// TIA Portal V19 export
DATA_BLOCK "GBL_TandD_DB"   // DB104
// stored: InstanceOfName GBL_TandD, InstanceOfType FB
"GBL_TandD"
   // VAR
   //    "write time" { ExternalAccessible := 'False'; ExternalVisible := 'False'; ExternalWritable := 'False'} : DTL;
   //    "System Time" { ExternalAccessible := 'False'; ExternalVisible := 'False'; ExternalWritable := 'False'} : DTL;
   // END_VAR
BEGIN
END_DATA_BLOCK
